(* PLC project Unnamed, Unknown Unnamed 1 *)
(* stored: creationDateTime 2026-02-02T16:50:47, modificationDateTime 2026-02-02T16:56:12 *)

PROGRAM program0
  VAR
    Fault_Active AT %M01 : BOOL;
    Cycle_Complete AT %M02 : BOOL;
    Buzzer AT %QX0.1 : BOOL;
  END_VAR

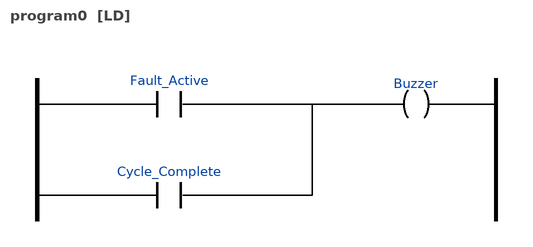
(* LD diagram, written out as Structured Text *)
Buzzer := Fault_Active OR Cycle_Complete;
END_PROGRAM

CONFIGURATION Config0
  RESOURCE Res0 ON PLC
    TASK task0(INTERVAL := T#20ms, PRIORITY := 0);
    PROGRAM instance0 WITH task0 : program0;
  END_RESOURCE
END_CONFIGURATION
